// TIA Portal V20 export
TYPE "zp_CITI_Configuration"
// stored: Namespace CITI_Logic
   STRUCT
      Instance : DInt;   // Map Instance
      UpdatePriority : DInt;   // Update Priority
      Features : "CITI_Logic.zp_CITI_Features";   // Features
      Parameters { S7_SetPoint := 'True'} : "CITI_Logic.zp_CITI_Parameters";   // Parameters
   END_STRUCT;
END_TYPE
